(* CoDeSys 2.3.9.41 project: twice-kns.pro *)
(* Libraries: STANDARD.LIB 4.10.05 10:14:46, IECSFC.LIB 13.4.06 14:51:28, SYSLIBTIME.LIB 20.2.06 13:31:16, SYSTASKINFO.LIB 20.2.06 13:31:38, ANALYZATION.LIB 5.10.99 08:05:06, SYSLIBCALLBACK.LIB 20.2.06 13:31:08 *)

(* PLC configuration (modules and I/O channels)
DI0_pmp1_auto AT %IX0.0 [BitInput]
DI1_pmp2_auto AT %IX0.1 [BitInput]
DI2_pmp1_man AT %IX0.2 [BitInput]
DI3_pmp2_man AT %IX0.3 [BitInput]
DI4_pmp1term AT %IX0.4 [BitInput]
DI5_pmp2term AT %IX0.5 [BitInput]
DO0_pmp1_turnOn AT %QX1.0 [BitOutput]
DO1_pmp2_turnOn AT %QX1.1 [BitOutput]
AT %QX1.2 [BitOutput]
AT %QX1.3 [BitOutput]
Special output [ID104] node 2, in %IB2 out %QB2 {Visibility = No; PinCount = 1}
  AT %QX2.0 [BitOutput] Special output
AI0_level_one AT %ID3.0 [FloatInput] Value
AT %IW3.1 [WordInput] Circular time
Analog Input [ID107] node 0, in %IB3.0 out %QB3.0
AI1_level_two AT %ID4.0 [FloatInput] Value
AT %IW4.1 [WordInput] Circular time
Analog Input [ID107] node 0, in %IB4.0 out %QB4.0
AT %ID5.0 [FloatInput] Value
AT %IW5.1 [WordInput] Circular time
Analog Input [ID107] node 0, in %IB5.0 out %QB5.0
AT %ID6.0 [FloatInput] Value
AT %IW6.1 [WordInput] Circular time
Analog Input [ID107] node 0, in %IB6.0 out %QB6.0
Analog output [ID106] node 7, in %IB7 out %QB7 {DAC_Type = Voltage 0-10 B; Analog_offset_correction = 0; Analog_full_range_correction = 0; SafeValueFloat = 0; Visibility = No}
  AT %QD7.0 [FloatOutput] Value
Analog output [ID106] node 8, in %IB8 out %QB8 {DAC_Type = Voltage 0-10 B; Analog_offset_correction = 0; Analog_full_range_correction = 0; SafeValueFloat = 0; Visibility = No}
  AT %QD8.0 [FloatOutput] Value
ModBus (Master) [MODBUS_MASTER_ID450] node 9, in %IB9 out %QB9 {Visibility = No}
  AT %QD9.0 [DWordOutput] Last address
  AT %QW9.1 [WordOutput] Last error
  RS-485-1 [COM1_USART] node 0, in %IB9.0 out %QB9.0 {CommunicationSpeed = 19200; Parity = NO PARITY CHECK; BitLength = 8 bits; StopLength = One stop bit; InterfaceType = RS485; FrameOriented = RTU; Timeout = 0; Visibility = No}
TCP [TCP_ID221] node 0, in %IB10.0.0 out %QB10.0.0 {RemotePort = 502; Visibility = No}
pan_TELEBITS AT %QW10.1.0 [WordOutput] pmp1run, pmp2run, pmp1term, pmp2term
pan_DISTBITS AT %QW10.2.0 [WordOutput] setTime, oneReset, twoReset
pan_oneLevel AT %QW10.3.0 [WordOutput]
pan_twoLevel AT %QW10.4.0 [WordOutput]
pan_onePres4ma AT %QW10.5.0 [WordOutput]
pan_onePres20ma AT %QW10.6.0 [WordOutput]
pan_twoPres4ma AT %QW10.7.0 [WordOutput]
pan_twoPres20ma AT %QW10.8.0 [WordOutput]
pan_oneUpp AT %QW10.9.0 [WordOutput]
pan_oneLww AT %QW10.10.0 [WordOutput]
pan_twoUpp AT %QW10.11.0 [WordOutput]
pan_twoLww AT %QW10.12.0 [WordOutput]
pan_pmp1_mode AT %QW10.13.0 [WordOutput] 0 - stop, 1 - auto, 2 - man
pan_pmp2_mode AT %QW10.14.0 [WordOutput]
pan_setMMin AT %QW10.15.0 [WordOutput]
pan_setHH AT %QW10.16.0 [WordOutput]
pan_setDD AT %QW10.17.0 [WordOutput]
pan_setMM AT %QW10.18.0 [WordOutput]
pan_setYYYY AT %QW10.19.0 [WordOutput]
pan_cursor AT %QW10.20.0 [WordOutput]
pan_aType_1 AT %QW10.21.0 [WordOutput]
pan_aTime_1 AT %QW10.22.0 [WordOutput]
pan_aDate_1 AT %QW10.23.0 [WordOutput]
pan_aOneLevel_1 AT %QW10.24.0 [WordOutput]
pan_aTwoLevel_1 AT %QW10.25.0 [WordOutput]
pan_aOneCurr_1 AT %QW10.26.0 [WordOutput]
pan_aTwoCurr_1 AT %QW10.27.0 [WordOutput]
pan_aType_2 AT %QW10.28.0 [WordOutput]
pan_aTime_2 AT %QW10.29.0 [WordOutput]
pan_aDate_2 AT %QW10.30.0 [WordOutput]
pan_aOneLevel_2 AT %QW10.31.0 [WordOutput]
pan_aTwoLevel_2 AT %QW10.32.0 [WordOutput]
pan_aOneCurr_2 AT %QW10.33.0 [WordOutput]
pan_aTwoCurr_2 AT %QW10.34.0 [WordOutput]
pan_aType_3 AT %QW10.35.0 [WordOutput]
pan_aTime_3 AT %QW10.36.0 [WordOutput]
pan_aDate_3 AT %QW10.37.0 [WordOutput]
pan_aOneLevel_3 AT %QW10.38.0 [WordOutput]
pan_aTwoLevel_3 AT %QW10.39.0 [WordOutput]
pan_aOneCurr_3 AT %QW10.40.0 [WordOutput]
pan_aTwoCurr_3 AT %QW10.41.0 [WordOutput]
pan_topPos AT %QW10.42.0 [WordOutput]
pan_midPos AT %QW10.43.0 [WordOutput]
pan_bottomPos AT %QW10.44.0 [WordOutput]
pan_pmp1state AT %QW10.45.0 [WordOutput] 0 - stop, 1 - run, 2 - blocked
pan_pmp2state AT %QW10.46.0 [WordOutput] 0 - stop, 1 - run, 2 - blocked
pan_HH AT %QW10.47.0 [WordOutput]
pan_MMin AT %QW10.48.0 [WordOutput]
pan_DD AT %QW10.49.0 [WordOutput]
pan_MM AT %QW10.50.0 [WordOutput]
pan_YYYY AT %QW10.51.0 [WordOutput]
*)

(* Global variable list: Global_Variables *)
VAR_GLOBAL
	(* Alarms *)
	Alarmy : WORD;

	oneSensBreak : BOOL; (* 1 *)
	oneSensShort : BOOL; (* 2 *)
	twoSensBreak : BOOL; (* 3 *)
	twoSensShort : BOOL; (* 4 *)
	oneTermal : BOOL; (* 5 *)
	twoTermal : BOOL; (* 6 *)


	(* Times *)
	GetTime: CurTimeEx;
	TimeAndDate: SystemTimeDate;
	Sys_Time: SysTime64;

END_VAR

(* POU PLC_PRG, ST *)
PROGRAM PLC_PRG
VAR
	NO_FIRST_PASS : BOOL := FALSE;

	(* one *)
	one_wPres4ma, one_wPres20ma : WORD;
	one_wLevel : WORD; (* текущмй уровень. точность 0.01 *)
	one_wUpp, one_wLww : WORD; (* верхний и нижний уровни. точность 0.01 *)
	one_pmpMustStart : BOOL;
	one_upperLevelReached : BOOL;
	one_lowerLevelReached : BOOL;

	(* two *)
	two_wPres4ma, two_wPres20ma : WORD;
	two_wLevel : WORD; (* текущий уровень. точность 0.01 *)
	two_wUpp, two_wLww : WORD; (* верхний и нижний уровни. точность 0.01 *)
	two_pmpMustStart : BOOL;
	two_upperLevelReached : BOOL;
	two_lowerLevelReached : BOOL;

	(* Times *)
	setTime : BOOL;

	(* Alarmes *)
	oneBreakDetect : BOOL;
	oneBreakTimer : TON;

	oneShortDetect : BOOL;
	oneShortTimer : TON;

	twoBreakDetect : BOOL;
	twoBreakTimer : TON;

	twoShortDetect : BOOL;
	twoShortTimer : TON;

	oneTermalDetect : BOOL;
	oneTermalTimer : TON;

	twoTermalDetect : BOOL;
	twoTermalTimer : TON;

	pmp1blocked, pmp2blocked : BOOL;
	oneBlockReset, twoBlockReset : BOOL;

END_VAR
VAR RETAIN
	(* one *)
	save_one_wPres4ma, save_one_wPres20ma : WORD;
	save_one_wUpp, save_one_wLww : WORD; (* верхний и нижний уровни. точность 0.01 *)

	(* two *)
	save_two_wPres4ma, save_two_wPres20ma : WORD;
	save_two_wUpp, save_two_wLww : WORD; (* верхний и нижний уровни. точность 0.01 *)

END_VAR
IF NO_FIRST_PASS = FALSE THEN
			WithdrawRetain;
			NO_FIRST_PASS := TRUE;
END_IF;

oneBlockReset := pan_DISTBITS.1;
twoBlockReset := pan_DISTBITS.2;

Times;

Alarmes;

ALARMS;

CheckNewVal;

Calibration;

ProcessOne;

ProcessTwo;

PumpsControl;

Forward;
END_PROGRAM
ACTION Alarmes:
(* ONE SENS BREAK *)
IF AI0_level_one < 3.7 THEN
	oneBreakDetect := TRUE;
ELSE
	oneBreakDetect := FALSE;
END_IF;

oneBreakTimer(IN:= oneBreakDetect, PT:=T#1s, Q=>oneSensBreak, ET=> );


(* ONE SENS SHORT *)
IF AI0_level_one > 21.0 THEN
	oneShortDetect := TRUE;
ELSE
	oneShortDetect := FALSE;
END_IF;

oneShortTimer(IN:= oneShortDetect, PT:=T#1s, Q=>oneSensShort, ET=> );


(* TWO SENS BREAK *)
IF AI1_level_two < 3.7 THEN
	twoBreakDetect := TRUE;
ELSE
	twoBreakDetect := FALSE;
END_IF;

twoBreakTimer(IN:= twoBreakDetect, PT:=T#1s, Q=>twoSensBreak, ET=> );


(* TWO SENS SHORT *)
IF AI1_level_two > 21.0 THEN
	twoShortDetect := TRUE;
ELSE
	twoShortDetect := FALSE;
END_IF;

twoShortTimer(IN:= twoShortDetect, PT:=T#1s, Q=>twoSensShort, ET=> );


(* ONE TERMAL *)
IF DI4_pmp1term = FALSE THEN
	oneTermalDetect := TRUE;
ELSE
	oneTermalDetect := FALSE;
END_IF;

oneTermalTimer(IN:= oneTermalDetect, PT:=T#1s, Q=>oneTermal, ET=> );

(* TWO TERMAL *)
IF DI5_pmp2term = FALSE THEN
	twoTermalDetect := TRUE;
ELSE
	twoTermalDetect := FALSE;
END_IF;

twoTermalTimer(IN:= twoTermalDetect, PT:=T#1s, Q=>twoTermal, ET=> );


(* ALARMY *)
Alarmy.0 := oneSensBreak;
Alarmy.1 := oneSensShort;
Alarmy.2 := twoSensBreak;
Alarmy.3 := twoSensShort;
Alarmy.4 := oneTermal;
Alarmy.5 := twoTermal;


IF oneSensBreak OR oneSensShort OR oneTermal THEN
	pmp1blocked := TRUE;
END_IF;

IF twoSensBreak OR twoSensShort OR twoTermal THEN
	pmp2blocked := TRUE;
END_IF;

IF oneBlockReset THEN
	pmp1blocked := FALSE;
	oneBlockReset := FALSE;
END_IF;

IF twoBlockReset THEN
	pmp2blocked := FALSE;
	twoBlockReset := FALSE;
END_IF;
END_ACTION
ACTION Calibration:
one_wLevel := one_wPres4ma  + ( REAL_TO_INT( AI0_level_one * 100 ) - 400 ) * ( one_wPres20ma - one_wPres4ma ) / 1600; (* wordpres := .... точность 0.01 *)

IF AI0_level_one < 4.0 THEN
	one_wLevel := 0;
END_IF;

two_wLevel := two_wPres4ma  + ( REAL_TO_INT( AI1_level_two * 100 ) - 400 ) * ( two_wPres20ma - two_wPres4ma ) / 1600; (* wordpres := .... точность 0.01 *)

IF AI1_level_two < 4.0 THEN
	two_wLevel := 0;
END_IF;
END_ACTION
ACTION CheckNewVal:
IF pan_onePres4ma <> one_wPres4ma THEN
	save_one_wPres4ma := pan_onePres4ma;
	one_wPres4ma := pan_onePres4ma;
END_IF;

IF pan_twoPres4ma <> two_wPres4ma THEN
	save_two_wPres4ma := pan_twoPres4ma;
	two_wPres4ma := pan_twoPres4ma;
END_IF;

IF pan_onePres20ma <> one_wPres20ma THEN
	save_one_wPres20ma := pan_onePres20ma;
	one_wPres20ma := pan_onePres20ma;
END_IF;

IF pan_twoPres20ma <> two_wPres20ma THEN
	save_two_wPres20ma := pan_twoPres20ma;
	two_wPres20ma := pan_twoPres20ma;
END_IF;

IF pan_oneLww <> one_wLww THEN
	save_one_wLww := pan_oneLww;
	one_wLww := pan_oneLww;
END_IF;

IF pan_twoLww <> two_wLww THEN
	save_two_wLww := pan_twoLww;
	two_wLww := pan_twoLww;
END_IF;

IF pan_oneUpp <> one_wUpp THEN
	save_one_wUpp := pan_oneUpp;
	one_wUpp := pan_oneUpp;
END_IF;

IF pan_twoUpp <> two_wUpp THEN
	save_two_wUpp := pan_twoUpp;
	two_wUpp := pan_twoUpp;
END_IF;
END_ACTION
ACTION Forward:
pan_oneLevel := one_wLevel;
pan_twoLevel := two_wLevel;

pan_TELEBITS.0 := DO0_pmp1_turnOn;
pan_TELEBITS.1 := DO1_pmp2_turnOn;
pan_TELEBITS.2 := DI4_pmp1term;
pan_TELEBITS.3 := DI5_pmp2term;


pan_HH := TimeAndDate.Hour;
pan_MMin := TimeAndDate.Minute;
pan_DD := TimeAndDate.Day;
pan_MM := TimeAndDate.Month;
pan_YYYY := TimeAndDate.Year;


IF Alarmy > 0 THEN
	pan_TELEBITS.4 := TRUE;
ELSE
	pan_TELEBITS.4 := FALSE;
END_IF;

IF DI0_pmp1_auto = FALSE AND DI2_pmp1_man = FALSE THEN
	pan_pmp1_mode := 0;
END_IF;

IF DI0_pmp1_auto = TRUE THEN
	pan_pmp1_mode := 1;
END_IF;

IF DI2_pmp1_man = TRUE THEN
	pan_pmp1_mode := 2;
END_IF;

IF DI1_pmp2_auto = FALSE AND DI3_pmp2_man = FALSE THEN
	pan_pmp2_mode := 0;
END_IF;

IF DI1_pmp2_auto = TRUE THEN
	pan_pmp2_mode := 1;
END_IF;

IF DI3_pmp2_man = TRUE THEN
	pan_pmp2_mode := 2;
END_IF;

IF  DO0_pmp1_turnOn THEN
	pan_pmp1state := 1;
ELSE
	pan_pmp1state := 0;
END_IF;

IF pmp1blocked THEN
	pan_pmp1state := 2;
END_IF;

IF  DO1_pmp2_turnOn THEN
	pan_pmp2state := 1;
ELSE
	pan_pmp2state := 0;
END_IF;

IF pmp2blocked THEN
	pan_pmp2state := 2;
END_IF;
END_ACTION
ACTION ProcessOne:
IF one_wLevel  > one_wUpp THEN
	one_upperLevelReached := TRUE;
ELSE
	one_upperLevelReached := FALSE;
END_IF;

IF one_wLevel > one_wLww THEN
	one_lowerLevelReached := TRUE;
ELSE
	one_lowerLevelReached := FALSE;
END_IF;

IF one_lowerLevelReached AND one_upperLevelReached THEN
	one_pmpMustStart := TRUE;
END_IF;

IF one_upperLevelReached = FALSE AND one_lowerLevelReached = FALSE THEN
	one_pmpMustStart := FALSE;
END_IF;
END_ACTION
ACTION ProcessTwo:
IF two_wLevel  > two_wUpp THEN
	two_upperLevelReached := TRUE;
ELSE
	two_upperLevelReached := FALSE;
END_IF;

IF two_wLevel > two_wLww THEN
	two_lowerLevelReached := TRUE;
ELSE
	two_lowerLevelReached := FALSE;
END_IF;

IF two_lowerLevelReached AND two_upperLevelReached THEN
	two_pmpMustStart := TRUE;
END_IF;

IF two_upperLevelReached = FALSE AND two_lowerLevelReached = FALSE THEN
	two_pmpMustStart := FALSE;
END_IF;
END_ACTION
ACTION PumpsControl:
IF ( DI0_pmp1_auto AND one_pmpMustStart ) OR DI2_pmp1_man THEN
	DO0_pmp1_turnOn := TRUE;
ELSE
	DO0_pmp1_turnOn := FALSE;
END_IF;

IF ( DI1_pmp2_auto AND two_pmpMustStart ) OR DI3_pmp2_man THEN
	DO1_pmp2_turnOn := TRUE;
ELSE
	DO1_pmp2_turnOn := FALSE;
END_IF;

IF DI0_pmp1_auto = FALSE AND DI2_pmp1_man = FALSE THEN
	DO0_pmp1_turnOn := FALSE;
END_IF;

IF DI1_pmp2_auto = FALSE AND DI3_pmp2_man = FALSE THEN
	DO1_pmp2_turnOn := FALSE;
END_IF;

IF pmp1blocked THEN
	DO0_pmp1_turnOn := FALSE;
END_IF;

IF pmp1blocked THEN
	DO1_pmp2_turnOn := FALSE;
END_IF;
END_ACTION
ACTION Times:
TimeAndDate.Day :=0;
TimeAndDate.DayOfWeek :=0;
TimeAndDate.dwHighMsec :=0;
TimeAndDate.dwLowMSecs :=0;
TimeAndDate.Milliseconds :=0;
TimeAndDate.Minute :=0;
TimeAndDate.Second :=0;
TimeAndDate.Hour :=0;
TimeAndDate.Year :=0;
TimeAndDate.Month :=0;
Sys_time.ulHigh :=0;
Sys_time.ulLow :=0;
GetTime (SystemTime:=Sys_Time , TimeDate:= TimeAndDate);


IF pan_DISTBITS.0 THEN
	TimeAndDate.Minute:=pan_setMMin;
	TimeAndDate.Second:=10;
	TimeAndDate.Hour:=pan_setHH;
	TimeAndDate.Day:=pan_setDD;
	TimeAndDate.Month:=pan_setMM;
	TimeAndDate.Year:=pan_setYYYY;
	GetTime (SystemTime:=Sys_Time , TimeDate:= TimeAndDate);

	pan_DISTBITS.0 := FALSE;
END_IF;
END_ACTION
ACTION WithdrawRetain:
pan_onePres4ma := save_one_wPres4ma;
pan_twoPres4ma :=  save_two_wPres4ma;

pan_onePres20ma := save_one_wPres20ma;
pan_twoPres20ma :=  save_two_wPres20ma;


pan_oneLww := save_one_wLww;
pan_twoLww :=  save_two_wLww;

pan_oneUpp := save_one_wUpp;
pan_twoUpp :=  save_two_wUpp;
END_ACTION

(* POU ALARMS, ST *)
PROGRAM ALARMS
VAR
	fp_oneSensBreak : BOOL; (* 1 *)
	fp_oneSensShort  : BOOL; (* 2 *)
	fp_twoSensBreak : BOOL; (* 3 *)
	fp_twoSensShort  : BOOL; (* 4 *)
	fp_oneTermal		: BOOL; (* 5 *)
	fp_twoTermal		: BOOL; (* 6 *)

	last_aType 	:  WORD;

	topPos, midPos, bottomPos : INT;

END_VAR
VAR RETAIN
	id	: INT;
	(* must be retain *)
	aType 		: ARRAY[0..99] OF WORD;
	aTime 		: ARRAY[0..99] OF WORD;
	aDate 		: ARRAY[0..99] OF WORD;
	oneLevel	: ARRAY[0..99] OF WORD;
	twoLevel	: ARRAY[0..99] OF WORD;
	oneCurr	: ARRAY[0..99] OF WORD;
	twoCurr	: ARRAY[0..99] OF WORD;

END_VAR
last_aType := 0;

IF pan_cursor = 127 THEN
	pan_cursor := INT_TO_WORD( id ) - 1;
END_IF

CorrectCursor;

FillFields;

Check;

pan_topPos := INT_TO_WORD( topPos );
pan_midPos := INT_TO_WORD( midPos );
pan_bottomPos := INT_TO_WORD( bottomPos );
END_PROGRAM
ACTION AddNew:
aType[ id ] := last_aType;
aTime[ id ] := TimeAndDate.Hour * 100 + TimeAndDate.Minute;
aDate[ id ] := TimeAndDate.Day * 100 + TimeAndDate.Month;
oneLevel[ id ] := pan_oneLevel;
twoLevel[ id ] := pan_twoLevel;
oneCurr[ id ] := 0;
twoCurr[ id ] := 0;

id := id + 1;

IF id >= 100 THEN
	id := 0;
END_IF;

pan_cursor := INT_TO_WORD( id );
END_ACTION
ACTION Check:
(* ONE SENS BREAK *)
IF oneSensBreak AND fp_oneSensBreak = FALSE THEN
	fp_onesensBreak := TRUE;
	last_aType := 1;
	AddNew;
END_IF;

IF oneSensBreak = FALSE THEN
	fp_oneSensBreak := FALSE;
END_IF;

(* ONE SENS SHORT *)
IF oneSensShort AND fp_oneSensShort = FALSE THEN
	fp_oneSensShort := TRUE;
	last_aType := 2;
	AddNew;
END_IF;

IF oneSensShort = FALSE THEN
	fp_oneSensShort := FALSE;
END_IF;


(* TWO SENS BREAK *)
IF twoSensBreak AND fp_twoSensBreak = FALSE THEN
	fp_twoSensBreak := TRUE;
	last_aType := 3;
	AddNew;
END_IF;

IF twoSensBreak = FALSE THEN
	fp_twoSensBreak := FALSE;
END_IF;

(* TWO SENS SHORT *)
IF twoSensShort AND fp_twoSensShort = FALSE THEN
	fp_twoSensShort := TRUE;
	last_aType := 4;
	AddNew;
END_IF;

IF twoSensShort = FALSE THEN
	fp_twoSensShort := FALSE;
END_IF;


(* ONE TERMAL *)
IF oneTermal AND fp_oneTermal = FALSE THEN
	fp_oneTermal := TRUE;
	last_aType := 5;
	AddNew;
END_IF;

IF oneTermal = FALSE THEN
	fp_oneTermal := FALSE;
END_IF;

(* TWO TERMAL *)
IF twoTermal AND fp_twoTermal = FALSE THEN
	fp_twoTermal := TRUE;
	last_aType := 6;
	AddNew;
END_IF;

IF twoTermal = FALSE THEN
	fp_twoTermal := FALSE;
END_IF;
END_ACTION
ACTION CorrectCursor:
IF pan_cursor > 99 THEN
	pan_cursor := 0;
END_IF;

topPos := pan_cursor;

midPos := pan_cursor - 1;

bottomPos := pan_cursor - 2;

IF pan_cursor = 0 THEN
	midPos := 99;
	bottomPos := 98;
END_IF;

IF pan_cursor = 1 THEN
	bottomPos := 99;
END_IF;
END_ACTION
ACTION FillFields:
pan_aType_1 			:= aType		[ topPos ];
pan_aTime_1 		:= aTime		[ topPos ];
pan_aDate_1 			:= aDate		[ topPos ];
pan_aOneLevel_1 	:= oneLevel	[ topPos ];
pan_aTwoLevel_1	:= twoLevel	[ topPos ];
pan_aOneLevel_1 	:= oneCurr		[ topPos ];
pan_aTwoLevel_1	:= twoCurr		[ topPos ];


pan_aType_2 			:= aType		[ midPos ];
pan_aTime_2 		:= aTime		[ midPos ];
pan_aDate_2			:= aDate		[ midPos ];
pan_aOneLevel_2 	:= oneLevel	[ midPos ];
pan_aTwoLevel_2 	:= twoLevel	[ midPos ];
pan_aOneCurr_2 		:= oneCurr		[ midPos ];
pan_aTwoCurr_2 		:= twoCurr		[ midPos ];


pan_aType_3 			:= aType		[ bottomPos ];
pan_aTime_3 		:= aTime		[ bottomPos ];
pan_aDate_3			:= aDate		[ bottomPos ];
pan_aOneLevel_3 	:= oneLevel	[ bottomPos ];
pan_aTwoLevel_3 	:= twoLevel	[ bottomPos ];
pan_aOneCurr_3 		:= oneCurr		[ bottomPos ];
pan_aTwoCurr_3 		:= twoCurr		[ bottomPos ];
END_ACTION
